FUNCTION_BLOCK FB_TCPIP
VAR_INPUT
	bNewItem				:BOOL;
	bConnectedRead			:BOOL;
	bConnectedWrite			:BOOL;
	bResetEANRegistry		:BOOL;
	ReadSocketHandler		:T_HSOCKET;
	WriteSocketHandler		:T_HSOCKET;
	iRead					:UINT;
	iWrite					:UINT;
END_VAR
VAR_OUTPUT
	aEANRegistry		:ARRAY[0..GVL_Constant.ITEM_ARRAY_SIZE] OF T_MaxString;
END_VAR
VAR
	sReadString				:T_MaxString;
	fbWrite					:FB_SocketSend;
	fbRead					:FB_SocketReceive;
	aWriteBytes				:ARRAY[0..1023] OF BYTE;
	aReadBytes				:ARRAY[0..1023] OF BYTE;
	nWriteLen				:UDINT;
	ReadComplete			:R_TRIG;
	tRefreshRead			:FB_ClockPulsDetailed;
	WriteSignal				:F_TRIG;
	i						:INT;
END_VAR

//Call Read & Write connected
A_TCPReading();
A_TCPWriting();

//Reset registry of EAN strings
IF PRG_Simulator.bStartGenerator OR PRG_Simulator.bStopGenerator OR (PRG_Simulator.i > PRG_Simulator.nTimeCount) OR bResetEANRegistry THEN
	FOR i := 0 TO GVL_Constant.ITEM_ARRAY_SIZE DO 
		aEANRegistry[i] := '';
	END_FOR

	iRead := 0;
	iWrite := 0;
	MEMSET(destAddr:=ADR(aReadBytes),fillByte:=0, n:=fbRead.nRecBytes);
	MEMSET(destAddr:=ADR(sReadString),fillByte:=0, n:=fbRead.nRecBytes);	
	
	
	//Reset commands
	bResetEANRegistry:=FALSE;
END_IF

ACTION A_TCPReading:
IF bConnectedRead THEN

	//Refresh read timer
	tRefreshRead(bEnable:=TRUE, tPulsLengthOn:=T#2MS, tPulsLengthOff:=T#2MS);
	
	fbRead(
		hSocket:=ReadSocketHandler, 
		cbLen:=SIZEOF(aReadBytes),
		pDest:=ADR(aReadBytes),
		bExecute:=tRefreshRead.bPuls);
		
	ReadComplete(CLK:=fbRead.nRecBytes > 0);
	
	
	//If byte read, copy into string.
	IF ReadComplete.Q THEN
		MEMCPY(destAddr:=ADR(sReadString), srcAddr:=ADR(aReadBytes),n:=fbRead.nRecBytes);
		aEANRegistry[iRead] := sReadString;
		MEMSET(destAddr:=ADR(aReadBytes),fillByte:=0, n:=fbRead.nRecBytes);
		MEMSET(destAddr:=ADR(sReadString),fillByte:=0, n:=fbRead.nRecBytes);
		iRead:=iRead+1;
	END_IF
END_IF;
END_ACTION

ACTION A_TCPWriting:
IF bConnectedWrite THEN	
	//Falling edge of item generator
	WriteSignal(CLK:=GVL_ItemSimulator.bSignalOut);
	
	IF WriteSignal.Q THEN
		//Get length of string written
		nWriteLen := INT_TO_UDINT(LEN(STR:=aEANRegistry[iWrite]));
	
		//Copy string into array of bytes
		MEMCPY(destAddr:=ADR(aWriteBytes),srcAddr:=ADR(aEANRegistry[iWrite]),n:=nWriteLen);
		iWrite := iWrite + 1;
	END_IF
		
	//Write byte array to TCP server
	fbWrite(
		hSocket:=WriteSocketHandler, 
		cbLen:=nWriteLen,
		pSrc:=ADR(aWriteBytes),
		bExecute:=WriteSignal.Q AND PRG_Simulator.stItemGenFromReg.bEnableGenerator);
END_IF;
END_ACTION

END_FUNCTION_BLOCK

(* stored: Version 1.1.0.1, ProductVersion 3.1.4024.12
   POU FB_TCPIP: Id {8a1361cc-b4d0-445e-95d0-5145c7c9d975}, SpecialFunc None
   Action A_TCPReading: Id {c6684671-51e7-43f4-84c9-10649b1f3710}
   Action A_TCPWriting: Id {a8da9708-cafa-4ccf-b159-6892f3e2e304} *)
